FUNCTION_BLOCK SimpleTimeChannel
VAR_INPUT
	EN: BOOL;
END_VAR
VAR_OUTPUT
	ENO: BOOL;
END_VAR
VAR
	LocalSystemTime: FB_LocalSystemTime;
	Active: BOOL;
	InitDone: bool;
END_VAR

IF NOT InitDone THEN
	EN := TRUE;
	InitDone := TRUE;
END_IF
LocalSystemTime(bEnable := TRUE);
IF LocalSystemTime.bValid THEN
	Active := (NOT EN) OR ((LocalSystemTime.systemTime.wHour > 5 AND LocalSystemTime.systemTime.wHour < 20) OR
		(LocalSystemTime.systemTime.wHour = 5 AND LocalSystemTime.systemTime.wMinute >= 30)); 
END_IF

ENO := EN AND Active;

END_FUNCTION_BLOCK

(* stored: Version 1.1.0.1, ProductVersion 3.1.4024.4
   POU SimpleTimeChannel: Id {e47102cb-d6a6-4acd-a377-83c30fec44bf}, SpecialFunc None *)
